TYPE ST_Point :
	STRUCT
		x : INT;
		y : INT;
	END_STRUCT
END_TYPE

(* stored: Version 1.1.0.1
   DUT ST_Point: Id {p} *)
